	REGION B1.14.1 Transfer Unit
	    //// Transfer B1.14.1
	    #"B1.14.1"(TransferID := _."B1.14.1",
	               TransferSensor:=_."ASiGW-MCC001-bw143-C2: Input"."LoadPresence -B1.14.1",
	               Fault := DB_UDI.ProductionLine.Fault.Stop.Conveyor[_."B1.14.1"],
	               Upstream := DB_UDI.ProductionLine.Upstream.Conveyor[_."B1.14.1"],
	               FrontSensor:=_."ASiGW-MCC001-bw143-C2: Input"."FrontSensor -B1.14.1",
	               EndSensor:=_."ASiGW-MCC001-bw143-C2: Input"."EndSensor -B1.14.1",
	               "Left/RightSensor":=_."ASiGW-MCC001-bw143-C2: Input"."LeftSensor -B1.14.1",
	               Downstream := DB_UDI.ProductionLine.DownstreamAccu.Stop.Conveyor[_."B1.14.1"],
	               TransferDirection := DB_ToteTracking.Conveyor[_."B1.14.1"].ToteDir,
	               StartSignal => _."ASiGW-MCC001-bw143-C2: Output"."StartSignal -B1.14.1",
	               Cmd1 => _."ASiGW-MCC001-bw143-C2: Output"."Command1 -B1.14.1",
	               Cmd2 => _."ASiGW-MCC001-bw143-C2: Output"."Command2 -B1.14.1",
	               ErrorReset => _."ASiGW-MCC001-bw143-C2: Output"."ErrorReset -B1.14.1");

	END_REGION

	REGION B1.15.1
	    //// B1.15.1 (Go straight TR_B1.17.1)
	    #"B1.15.1"(ConveyorID := _."B1.15.1",
	               ConveyorSensor:=_."ASiGW-MCC001-bw143-C2: Input"."Sensor B1.15.1",
	               Fault := DB_UDI.ProductionLine.Fault.Stop.Conveyor[_."B1.15.1"],
	               Upstream := DB_UDI.ProductionLine.Upstream.Conveyor[_."B1.15.1"],
	               Downstream := DB_UDI.ProductionLine.DownstreamAccu.Stop.Conveyor[_."B1.15.1"],
	               Interlock := DB_UDI.ProductionLine.Interlock.Stop.Conveyor[_."B1.15.1"],
	               RunForward=>_."ASiGW-MCC001-bw143-C2: Output"."Motor B1.15.1",
	               WriteAsiDir=>_."ASiGW-MCC001-bw143-C2: Output"."Dir B1.15.1");

	END_REGION

	REGION B1.15.2
	    //B1.15.2
	    #"B1.15.2"(ConveyorID := _."B1.15.2",
	               ConveyorSensor:=_."ASiGW-MCC001-bw143-C2: Input"."Sensor B1.15.2",
	               Fault := DB_UDI.ProductionLine.Fault.Stop.Conveyor[_."B1.15.2"],
	               Upstream := DB_UDI.ProductionLine.Upstream.Conveyor[_."B1.15.2"],
	               Downstream := DB_UDI.ProductionLine.DownstreamAccu.Stop.Conveyor[_."B1.15.2"],
	               Interlock := DB_UDI.ProductionLine.Interlock.Stop.Conveyor[_."B1.15.2"],
	               RunForward=>_."ASiGW-MCC001-bw143-C2: Output"."Motor B1.15.2",
	               WriteAsiDir=>_."ASiGW-MCC001-bw143-C2: Output"."Dir B1.15.2");

	END_REGION

	REGION B1.16.1
	    //B1.16.1
	    #"B1.16.1"(ConveyorID := _."B1.16.1",
	               ConveyorSensor:=_."ASiGW-MCC001-bw143-C2: Input"."Sensor B1.16.8",
	               Fault := DB_UDI.ProductionLine.Fault.Stop.Conveyor[_."B1.16.1"],
	               Upstream := DB_UDI.ProductionLine.Upstream.Conveyor[_."B1.16.1"],
	               Downstream := DB_UDI.ProductionLine.DownstreamAccu.Stop.Conveyor[_."B1.16.1"],
	               Interlock := DB_UDI.ProductionLine.Interlock.Stop.Conveyor[_."B1.16.1"],
	               RunForward => _."ASiGW-MCC001-bw143-C2: Output"."Motor B1.16.1",
	               WriteAsiDir => _."ASiGW-MCC001-bw143-C2: Output"."Dir B1.16.1");

	END_REGION

	REGION B1.16.2
	    //B1.16.2
	    #"B1.16.2"(ConveyorID := _."B1.16.2",
	               ConveyorSensor:=_."ASiGW-MCC001-bw143-C2: Input"."Sensor B1.16.8",
	               Fault := DB_UDI.ProductionLine.Fault.Stop.Conveyor[_."B1.16.2"],
	               Upstream := DB_UDI.ProductionLine.Upstream.Conveyor[_."B1.16.2"],
	               Downstream := DB_UDI.ProductionLine.DownstreamAccu.Stop.Conveyor[_."B1.16.2"],
	               Interlock := DB_UDI.ProductionLine.Interlock.Stop.Conveyor[_."B1.16.2"],
	               RunForward=>_."ASiGW-MCC001-bw143-C2: Output"."Motor B1.16.2",
	               WriteAsiDir=>_."ASiGW-MCC001-bw143-C2: Output"."Dir B1.16.2");

	END_REGION

	REGION B1.16.3
	    //B1.16.3
	    #"B1.16.3"(ConveyorID := _."B1.16.3",
	               ConveyorSensor:=_."ASiGW-MCC001-bw143-C2: Input"."Sensor B1.16.8",
	               Fault := DB_UDI.ProductionLine.Fault.Stop.Conveyor[_."B1.16.3"],
	               Upstream := DB_UDI.ProductionLine.Upstream.Conveyor[_."B1.16.3"],
	               Downstream := DB_UDI.ProductionLine.DownstreamAccu.Stop.Conveyor[_."B1.16.3"],
	               Interlock := DB_UDI.ProductionLine.Interlock.Stop.Conveyor[_."B1.16.3"],
	               RunForward=>_."ASiGW-MCC001-bw143-C2: Output"."Motor B1.16.3",
	               WriteAsiDir=>_."ASiGW-MCC001-bw143-C2: Output"."Dir B1.16.3");

	END_REGION

	REGION B1.16.4
	    //B1.16.4
	    #"B1.16.4"(ConveyorID := _."B1.16.4",
	               ConveyorSensor:=_."ASiGW-MCC001-bw143-C2: Input"."Sensor B1.16.8",
	               Fault := DB_UDI.ProductionLine.Fault.Stop.Conveyor[_."B1.16.4"],
	               Upstream := DB_UDI.ProductionLine.Upstream.Conveyor[_."B1.16.4"],
	               Downstream := DB_UDI.ProductionLine.DownstreamAccu.Stop.Conveyor[_."B1.16.4"],
	               Interlock := DB_UDI.ProductionLine.Interlock.Stop.Conveyor[_."B1.16.4"],
	               RunForward=>_."ASiGW-MCC001-bw143-C2: Output"."Motor B1.16.4",
	               WriteAsiDir=>_."ASiGW-MCC001-bw143-C2: Output"."Dir B1.16.4");

	END_REGION

	REGION B1.16.5
	    //B1.16.5
	    #"B1.16.5"(ConveyorID := _."B1.16.5",
	               ConveyorSensor:=_."ASiGW-MCC001-bw143-C2: Input"."Sensor B1.16.8",
	               Fault := DB_UDI.ProductionLine.Fault.Stop.Conveyor[_."B1.16.5"],
	               Upstream := DB_UDI.ProductionLine.Upstream.Conveyor[_."B1.16.5"],
	               Downstream := DB_UDI.ProductionLine.DownstreamAccu.Stop.Conveyor[_."B1.16.5"],
	               Interlock := DB_UDI.ProductionLine.Interlock.Stop.Conveyor[_."B1.16.5"],
	               RunForward=>_."ASiGW-MCC001-bw143-C2: Output"."Motor B1.16.5",
	               WriteAsiDir=>_."ASiGW-MCC001-bw143-C2: Output"."Dir B1.16.5");

	END_REGION

	REGION B1.16.6
	    //B1.16.6
	    #"B1.16.6"(ConveyorID := _."B1.16.6",
	               ConveyorSensor:=_."ASiGW-MCC001-bw143-C2: Input"."Sensor B1.16.8",
	               Fault := DB_UDI.ProductionLine.Fault.Stop.Conveyor[_."B1.16.6"],
	               Upstream := DB_UDI.ProductionLine.Upstream.Conveyor[_."B1.16.6"],
	               Downstream := DB_UDI.ProductionLine.DownstreamAccu.Stop.Conveyor[_."B1.16.6"],
	               Interlock := DB_UDI.ProductionLine.Interlock.Stop.Conveyor[_."B1.16.6"],
	               RunForward=>_."ASiGW-MCC001-bw143-C2: Output"."Motor B1.16.6",
	               WriteAsiDir=>_."ASiGW-MCC001-bw143-C2: Output"."Dir B1.16.6");

	END_REGION

	REGION B1.16.7
	    //B1.16.7
	    #"B1.16.7"(ConveyorID := _."B1.16.7",
	               ConveyorSensor:=_."ASiGW-MCC001-bw143-C2: Input"."Sensor B1.16.8",
	               Fault := DB_UDI.ProductionLine.Fault.Stop.Conveyor[_."B1.16.7"],
	               Upstream := DB_UDI.ProductionLine.Upstream.Conveyor[_."B1.16.7"],
	               Downstream := DB_UDI.ProductionLine.DownstreamAccu.Stop.Conveyor[_."B1.16.7"],
	               Interlock := DB_UDI.ProductionLine.Interlock.Stop.Conveyor[_."B1.16.7"],
	               RunForward => _."ASiGW-MCC001-bw143-C2: Output"."Motor B1.16.7",
	               WriteAsiDir => _."ASiGW-MCC001-bw143-C2: Output"."Dir B1.16.7");

	END_REGION

	REGION B1.16.8
	    //B1.16.8
	    #"B1.16.8"(ConveyorID := _."B1.16.8",
	               ConveyorSensor:=_."ASiGW-MCC001-bw143-C2: Input"."Sensor B1.16.8",
	               Fault := DB_UDI.ProductionLine.Fault.Stop.Conveyor[_."B1.16.8"],
	               Upstream := DB_UDI.ProductionLine.Upstream.Conveyor[_."B1.16.8"],
	               Downstream := DB_UDI.ProductionLine.DownstreamAccu.Stop.Conveyor[_."B1.16.8"],
	               Interlock := DB_UDI.ProductionLine.Interlock.Stop.Conveyor[_."B1.16.8"],
	               RunForward=>_."ASiGW-MCC001-bw143-C2: Output"."Motor B1.16.8",
	               WriteAsiDir=>_."ASiGW-MCC001-bw143-C2: Output"."Dir B1.16.8");

	END_REGION

	REGION B1.17.1
	    //// B1.17.1 (DP3)
	    #"B1.17.1"(ConveyorID := _."B1.17.1",
	               ConveyorSensor:=_."ASiGW-MCC001-bw143-C2: Input"."Sensor B1.17.1",
	               Fault := DB_UDI.ProductionLine.Fault.Stop.Conveyor[_."B1.17.1"],
	               Upstream := DB_UDI.ProductionLine.Upstream.Conveyor[_."B1.17.1"],
	               Downstream := DB_UDI.ProductionLine.DownstreamAccu.Stop.Conveyor[_."B1.17.1"],
	               Interlock := DB_UDI.ProductionLine.Interlock.Stop.Conveyor[_."B1.17.1"],
	               RunForward => _."ASiGW-MCC001-bw143-C2: Output"."Motor B1.17.1",
	               WriteAsiDir => _."ASiGW-MCC001-bw143-C2: Output"."Dir B1.17.1");

	END_REGION

	REGION B1.17.2
	    //B1.17.2
	    #"B1.17.2"(ConveyorID := _."B1.17.2",
	               ConveyorSensor:=_."ASiGW-MCC001-bw143-C2: Input"."Sensor B1.17.2",
	               Fault := DB_UDI.ProductionLine.Fault.Stop.Conveyor[_."B1.17.2"],
	               Upstream := DB_UDI.ProductionLine.Upstream.Conveyor[_."B1.17.2"],
	               Downstream := DB_UDI.ProductionLine.DownstreamAccu.Stop.Conveyor[_."B1.17.2"],
	               Interlock := DB_UDI.ProductionLine.Interlock.Stop.Conveyor[_."B1.17.2"],
	               RunForward => _."ASiGW-MCC001-bw143-C2: Output"."Motor B1.17.2",
	               WriteAsiDir => _."ASiGW-MCC001-bw143-C2: Output"."Dir B1.17.2");

	END_REGION

	REGION B1.17.3
	    //B1.17.3
	    #"B1.17.3"(ConveyorID := _."B1.17.3",
	               ConveyorSensor:=_."ASiGW-MCC001-bw143-C2: Input"."Sensor B1.17.3",
	               Fault := DB_UDI.ProductionLine.Fault.Stop.Conveyor[_."B1.17.3"],
	               Upstream := DB_UDI.ProductionLine.Upstream.Conveyor[_."B1.17.3"],
	               Downstream := DB_UDI.ProductionLine.DownstreamAccu.Stop.Conveyor[_."B1.17.3"],
	               Interlock := DB_UDI.ProductionLine.Interlock.Stop.Conveyor[_."B1.17.3"],
	               RunForward => _."ASiGW-MCC001-bw143-C2: Output"."Motor B1.17.3",
	               WriteAsiDir => _."ASiGW-MCC001-bw143-C2: Output"."Dir B1.17.3");

	END_REGION

	REGION B1.17.4
	    //B1.17.4
	    #"B1.17.4"(ConveyorID := _."B1.17.4",
	               ConveyorSensor:=_."ASiGW-MCC001-bw143-C2: Input"."Sensor B1.17.4",
	               Fault := DB_UDI.ProductionLine.Fault.Stop.Conveyor[_."B1.17.4"],
	               Upstream := DB_UDI.ProductionLine.Upstream.Conveyor[_."B1.17.4"],
	               Downstream := DB_UDI.ProductionLine.DownstreamAccu.Stop.Conveyor[_."B1.17.4"],
	               Interlock := DB_UDI.ProductionLine.Interlock.Stop.Conveyor[_."B1.17.4"],
	               RunForward => _."ASiGW-MCC001-bw143-C2: Output"."Motor B1.17.4",
	               WriteAsiDir => _."ASiGW-MCC001-bw143-C2: Output"."Dir B1.17.4");

	END_REGION

	REGION B1.18.1 Transfer Unit
	    //// Transfer B1.18.1
	    #"B1.18.1"(TransferID := _."B1.18.1",
	               TransferSensor:=_."ASiGW-MCC001-bw143-C2: Input"."LoadPresence -B1.18.1",
	               Fault := DB_UDI.ProductionLine.Fault.Stop.Conveyor[_."B1.18.1"],
	               Upstream := DB_UDI.ProductionLine.Upstream.Conveyor[_."B1.18.1"],
	               FrontSensor:=_."ASiGW-MCC001-bw143-C2: Input"."FrontSensor -B1.18.1",
	               EndSensor:=_."ASiGW-MCC001-bw143-C2: Input"."EndSensor -B1.18.1",
	               "Left/RightSensor":=_."ASiGW-MCC001-bw143-C2: Input"."LeftSensor -B1.18.1",
	               Downstream := DB_UDI.ProductionLine.DownstreamAccu.Stop.Conveyor[_."B1.18.1"],
	               TransferDirection := DB_ToteTracking.Conveyor[_."B1.18.1"].ToteDir,
	               StartSignal => _."ASiGW-MCC001-bw143-C2: Output"."StartSignal -B1.18.1",
	               Cmd1 => _."ASiGW-MCC001-bw143-C2: Output"."Command1 -B1.18.1",
	               Cmd2 => _."ASiGW-MCC001-bw143-C2: Output"."Command2 -B1.18.1",
	               ErrorReset => _."ASiGW-MCC001-bw143-C2: Output"."ErrorReset -B1.18.1");

	END_REGION

	REGION B1.19.1
	    //B1.19.1
	    #"B1.19.1"(ConveyorID := _."B1.19.1",
	               ConveyorSensor:=_."ASiGW-MCC001-bw143-C2: Input"."Sensor B1.19.1",
	               Fault := DB_UDI.ProductionLine.Fault.Stop.Conveyor[_."B1.19.1"],
	               Upstream := DB_UDI.ProductionLine.Upstream.Conveyor[_."B1.19.1"],
	               Downstream := DB_UDI.ProductionLine.DownstreamAccu.Stop.Conveyor[_."B1.19.1"],
	               Interlock := DB_UDI.ProductionLine.Interlock.Stop.Conveyor[_."B1.19.1"],
	               RunForward => _."ASiGW-MCC001-bw143-C2: Output"."Motor B1.19.1",
	               WriteAsiDir => _."ASiGW-MCC001-bw143-C2: Output"."Dir B1.19.1");

	END_REGION

	REGION B1.20.1
	    //B1.20.1
	    #"B1.20.1"(ConveyorID := _."B1.20.1",
	               ConveyorSensor:=_."ASiGW-MCC001-bw143-C2: Input"."Sensor B1.20.1",
	               Fault := DB_UDI.ProductionLine.Fault.Stop.Conveyor[_."B1.20.1"],
	               Upstream := DB_UDI.ProductionLine.Upstream.Conveyor[_."B1.20.1"],
	               Downstream := DB_UDI.ProductionLine.DownstreamAccu.Stop.Conveyor[_."B1.20.1"],
	               Interlock := DB_UDI.ProductionLine.Interlock.Stop.Conveyor[_."B1.20.1"],
	               RunForward => _."ASiGW-MCC001-bw143-C2: Output"."Motor B1.20.1",
	               WriteAsiDir => _."ASiGW-MCC001-bw143-C2: Output"."Dir B1.20.1");

	END_REGION

	REGION B1.20.2
	    //B1.20.2
	    #"B1.20.2"(ConveyorID := _."B1.20.2",
	               ConveyorSensor:=_."ASiGW-MCC001-bw143-C2: Input"."Sensor B1.20.2",
	               Fault := DB_UDI.ProductionLine.Fault.Stop.Conveyor[_."B1.20.2"],
	               Upstream := DB_UDI.ProductionLine.Upstream.Conveyor[_."B1.20.2"],
	               Downstream := DB_UDI.ProductionLine.DownstreamAccu.Stop.Conveyor[_."B1.20.2"],
	               Interlock := DB_UDI.ProductionLine.Interlock.Stop.Conveyor[_."B1.20.2"],
	               RunForward => _."ASiGW-MCC001-bw143-C2: Output"."Motor B1.20.2",
	               WriteAsiDir => _."ASiGW-MCC001-bw143-C2: Output"."Dir B1.20.2");

	END_REGION

	REGION B1.21.1
	    //B1.21.1
	    #"B1.21.1"(ConveyorID := _."B1.21.1",
	               ConveyorSensor:=_."ASiGW-MCC001-bw143-C2: Input"."Sensor B1.21.1",
	               Fault := DB_UDI.ProductionLine.Fault.Stop.Conveyor[_."B1.21.1"],
	               Upstream := DB_UDI.ProductionLine.Upstream.Conveyor[_."B1.21.1"],
	               Downstream := DB_UDI.ProductionLine.DownstreamAccu.Stop.Conveyor[_."B1.21.1"],
	               Interlock := DB_UDI.ProductionLine.Interlock.Stop.Conveyor[_."B1.21.1"],
	               RunForward => _."ASiGW-MCC001-bw143-C2: Output"."Motor B1.21.1",
	               WriteAsiDir => _."ASiGW-MCC001-bw143-C2: Output"."Dir B1.21.1");

	END_REGION

	REGION B1.21.2
	    //B1.21.2
	    #"B1.21.2"(ConveyorID := _."B1.21.2",
	               ConveyorSensor:=_."ASiGW-MCC001-bw143-C2: Input"."Sensor B1.21.2",
	               Fault := DB_UDI.ProductionLine.Fault.Stop.Conveyor[_."B1.21.2"],
	               Upstream := DB_UDI.ProductionLine.Upstream.Conveyor[_."B1.21.2"],
	               Downstream := DB_UDI.ProductionLine.DownstreamAccu.Stop.Conveyor[_."B1.21.2"],
	               Interlock := DB_UDI.ProductionLine.Interlock.Stop.Conveyor[_."B1.21.2"],
	               RunForward => _."ASiGW-MCC001-bw143-C2: Output"."Motor B1.21.2",
	               WriteAsiDir => _."ASiGW-MCC001-bw143-C2: Output"."Dir B1.21.2");

	END_REGION

	REGION B1.21.3
	    //B1.21.3
	    #"B1.21.3"(ConveyorID := _."B1.21.3",
	               ConveyorSensor:=_."ASiGW-MCC001-bw143-C2: Input"."Sensor B1.23.1",
	               Fault := DB_UDI.ProductionLine.Fault.Stop.Conveyor[_."B1.21.3"],
	               Upstream := DB_UDI.ProductionLine.Upstream.Conveyor[_."B1.21.3"],
	               Downstream := DB_UDI.ProductionLine.DownstreamAccu.Stop.Conveyor[_."B1.21.3"],
	               Interlock := DB_UDI.ProductionLine.Interlock.Stop.Conveyor[_."B1.21.3"],
	               RunForward => _."ASiGW-MCC001-bw143-C2: Output"."Motor B1.21.3",
	               WriteAsiDir => _."ASiGW-MCC001-bw143-C2: Output"."Dir B1.21.3");

	END_REGION

	REGION B1.22.1
	    //B1.22.1
	    #"B1.22.1"(ConveyorID := _."B1.22.1",
	               ConveyorSensor:=_."ASiGW-MCC001-bw143-C2: Input"."Sensor B1.23.1",
	               Fault := DB_UDI.ProductionLine.Fault.Stop.Conveyor[_."B1.22.1"],
	               Upstream := DB_UDI.ProductionLine.Upstream.Conveyor[_."B1.22.1"],
	               Downstream := DB_UDI.ProductionLine.DownstreamAccu.Stop.Conveyor[_."B1.22.1"],
	               Interlock := DB_UDI.ProductionLine.Interlock.Stop.Conveyor[_."B1.22.1"],
	               RunForward => _."ASiGW-MCC001-bw143-C2: Output"."Motor - B1.22.1",
	               WriteAsiDir => _."ASiGW-MCC001-bw143-C2: Output"."2-30A Dir",
	               WriteAsiSpeed => _."ASiGW-MCC001-bw143-C2: Output"."2-30A Speed");

	END_REGION

	REGION B1.23.1
	    ////B1.23.1 Arm for Merger1
	    #"B1.23.1"(ConveyorID := _."B1.23.1",
	               ConveyorSensor:=_."ASiGW-MCC001-bw143-C2: Input"."Sensor B1.23.1",
	               Fault := DB_UDI.ProductionLine.Fault.Stop.Conveyor[_."B1.23.1"],
	               Upstream := DB_UDI.ProductionLine.Upstream.Conveyor[_."B1.23.1"],
	               Downstream := DB_UDI.ProductionLine.DownstreamAccu.Stop.Conveyor[_."B1.23.1"],
	               Interlock := DB_UDI.ProductionLine.Interlock.Stop.Conveyor[_."B1.23.1"],
	               RunForward => _."ASiGW-MCC001-bw143-C2: Output"."Motor B1.23.1",
	               WriteAsiDir => _."ASiGW-MCC001-bw143-C2: Output"."Dir B1.23.1");

	END_REGION

	REGION C1.3.1 Transfer Unit
	    ////Transfer C1.3.1
	    #"C1.3.1"(TransferID := _."C1.3.1",
	              TransferSensor:=_."ASiGW-MCC001-bw143-C2: Input"."LoadPresence -C1.3.1",
	              Fault := DB_UDI.ProductionLine.Fault.Stop.Conveyor[_."C1.3.1"],
	              Upstream := DB_UDI.ProductionLine.Upstream.Conveyor[_."C1.3.1"],
	              FrontSensor:=_."ASiGW-MCC001-bw143-C2: Input"."FrontSensor -C1.3.1",
	              EndSensor:=_."ASiGW-MCC001-bw143-C2: Input"."EndSensor -C1.3.1",
	              "Left/RightSensor":=_."ASiGW-MCC001-bw143-C2: Input"."LeftSensor -C1.3.1",
	              Downstream := DB_UDI.ProductionLine.DownstreamAccu.Stop.Conveyor[_."C1.3.1"],
	              TransferDirection := DB_ToteTracking.Conveyor[_."C1.3.1"].ToteDir,
	              StartSignal => _."ASiGW-MCC001-bw143-C2: Output"."StartSignal -C1.3.1",
	              Cmd1 => _."ASiGW-MCC001-bw143-C2: Output"."Command1 -C1.3.1",
	              Cmd2 => _."ASiGW-MCC001-bw143-C2: Output"."Command2 -C1.3.1",
	              ErrorReset => _."ASiGW-MCC001-bw143-C2: Output"."ErrorReset -C1.3.1");

	END_REGION

	REGION C1.2.2
	    //// C1.2.2  (Go Right TR_C1.1.3)
	    #"C1.2.2"(ConveyorID := _."C1.2.2",
	              ConveyorSensor:=_."ASiGW-MCC001-bw143-C2: Input"."Sensor C1.2.2",
	              Fault := DB_UDI.ProductionLine.Fault.Stop.Conveyor[_."C1.2.2"],
	              Upstream := DB_UDI.ProductionLine.Upstream.Conveyor[_."C1.2.2"],
	              Downstream := DB_UDI.ProductionLine.DownstreamAccu.Stop.Conveyor[_."C1.2.2"],
	              Interlock := DB_UDI.ProductionLine.Interlock.Stop.Conveyor[_."C1.2.2"],
	              RunForward=>_."ASiGW-MCC001-bw143-C2: Output"."Motor C1.2.2",
	              WriteAsiDir=>_."ASiGW-MCC001-bw143-C2: Output"."Dir C1.2.2");

	END_REGION

	REGION C1.2.1
	    //C1.2.1
	    #"C1.2.1"(ConveyorID := _."C1.2.1",
	              ConveyorSensor:=_."ASiGW-MCC001-bw143-C2: Input"."Sensor C1.2.1",
	              Fault := DB_UDI.ProductionLine.Fault.Stop.Conveyor[_."C1.2.1"],
	              Upstream := DB_UDI.ProductionLine.Upstream.Conveyor[_."C1.2.1"],
	              Downstream := DB_UDI.ProductionLine.DownstreamAccu.Stop.Conveyor[_."C1.2.1"],
	              Interlock := DB_UDI.ProductionLine.Interlock.Stop.Conveyor[_."C1.2.1"],
	              RunForward=>_."ASiGW-MCC001-bw143-C2: Output"."Motor C1.2.1",
	              WriteAsiDir=>_."ASiGW-MCC001-bw143-C2: Output"."Dir C1.2.1");

	END_REGION

	REGION C1.4.1
	    //// C1.4.1  (Go Left TR_C1.1.3)
	    #"C1.4.1"(ConveyorID := _."C1.4.1",
	              ConveyorSensor:=_."ASiGW-MCC001-bw143-C2: Input"."Sensor C1.4.1",
	              Fault := DB_UDI.ProductionLine.Fault.Stop.Conveyor[_."C1.4.1"],
	              Upstream := DB_UDI.ProductionLine.Upstream.Conveyor[_."C1.4.1"],
	              Downstream := DB_UDI.ProductionLine.DownstreamAccu.Stop.Conveyor[_."C1.4.1"],
	              Interlock := DB_UDI.ProductionLine.Interlock.Stop.Conveyor[_."C1.4.1"],
	              RunForward=>_."ASiGW-MCC001-bw143-C2: Output"."Motor C1.4.1",
	              WriteAsiDir=>_."ASiGW-MCC001-bw143-C2: Output"."Dir C1.4.1");

	END_REGION

	REGION C1.4.2
	    //C1.4.2
	    #"C1.4.2"(ConveyorID := _."C1.4.2",
	              ConveyorSensor:=_."ASiGW-MCC001-bw143-C2: Input"."Sensor C1.4.2",
	              Fault := DB_UDI.ProductionLine.Fault.Stop.Conveyor[_."C1.4.2"],
	              Upstream := DB_UDI.ProductionLine.Upstream.Conveyor[_."C1.4.2"],
	              Downstream := DB_UDI.ProductionLine.DownstreamAccu.Stop.Conveyor[_."C1.4.2"],
	              Interlock := DB_UDI.ProductionLine.Interlock.Stop.Conveyor[_."C1.4.2"],
	              RunForward=>_."ASiGW-MCC001-bw143-C2: Output"."Motor C1.4.2",
	              WriteAsiDir=>_."ASiGW-MCC001-bw143-C2: Output"."Dir C1.4.2");

	END_REGION

	REGION D1.1.1
	    ////  D1.1.1 (Go Right DP4)
	    #"D1.1.1"(ConveyorID := _."D1.1.1",
	              ConveyorSensor:=_."ASiGW-MCC001-bw200-C1: Input"."Sensor D1.2.1",
	              Fault := DB_UDI.ProductionLine.Fault.Stop.Conveyor[_."D1.1.1"],
	              Upstream := DB_UDI.ProductionLine.Upstream.Conveyor[_."D1.1.1"],
	              Downstream := DB_UDI.ProductionLine.DownstreamAccu.Stop.Conveyor[_."D1.1.1"],
	              Interlock := DB_UDI.ProductionLine.Interlock.Stop.Conveyor[_."D1.1.1"],
	              RunForward=>_."ASiGW-MCC001-bw200-C1: Output"."Motor D1.1.1",
	              WriteAsiDir=>_."ASiGW-MCC001-bw200-C1: Output"."Dir D1.1.1");

	END_REGION

	REGION D1.2.1
	    //D1.2.1
	    #"D1.2.1"(ConveyorID := _."D1.2.1",
	              ConveyorSensor:=_."ASiGW-MCC001-bw200-C1: Input"."Sensor D1.2.1",
	              Fault := DB_UDI.ProductionLine.Fault.Stop.Conveyor[_."D1.2.1"],
	              Upstream := DB_UDI.ProductionLine.Upstream.Conveyor[_."D1.2.1"],
	              Downstream := DB_UDI.ProductionLine.DownstreamAccu.Stop.Conveyor[_."D1.2.1"],
	              Interlock := DB_UDI.ProductionLine.Interlock.Stop.Conveyor[_."D1.2.1"],
	              RunForward=>_."ASiGW-MCC001-bw200-C1: Output"."Motor - D1.2.1",
	              WriteAsiDir=>_."ASiGW-MCC001-bw200-C1: Output"."1-2A Dir",
	              WriteAsiSpeed=>_."ASiGW-MCC001-bw200-C1: Output"."1-2A Speed");

	END_REGION

	REGION D1.3.1
	    //D1.3.1
	    #"D1.3.1"(ConveyorID := _."D1.3.1",
	              ConveyorSensor:=_."ASiGW-MCC001-bw200-C1: Input"."Sensor D1.3.1",
	              Fault := DB_UDI.ProductionLine.Fault.Stop.Conveyor[_."D1.3.1"],
	              Upstream := DB_UDI.ProductionLine.Upstream.Conveyor[_."D1.3.1"],
	              Downstream := DB_UDI.ProductionLine.DownstreamAccu.Stop.Conveyor[_."D1.3.1"],
	              Interlock := DB_UDI.ProductionLine.Interlock.Stop.Conveyor[_."D1.3.1"],
	              RunForward=>_."ASiGW-MCC001-bw200-C1: Output"."Motor - D1.3.1",
	              WriteAsiDir=>_."ASiGW-MCC001-bw200-C1: Output"."1-2A Dir",
	              WriteAsiSpeed=>_."ASiGW-MCC001-bw200-C1: Output"."1-2A Speed");

	END_REGION

	REGION D1.4.1
	    //D1.4.1
	    #"D1.4.1"(ConveyorID := _."D1.4.1",
	              ConveyorSensor:=_."ASiGW-MCC001-bw200-C1: Input"."Sensor D1.4.1",
	              Fault := DB_UDI.ProductionLine.Fault.Stop.Conveyor[_."D1.4.1"],
	              Upstream := DB_UDI.ProductionLine.Upstream.Conveyor[_."D1.4.1"],
	              Downstream := DB_UDI.ProductionLine.DownstreamAccu.Stop.Conveyor[_."D1.4.1"],
	              Interlock := DB_UDI.ProductionLine.Interlock.Stop.Conveyor[_."D1.4.1"],
	              RunForward=>_."ASiGW-MCC001-bw200-C1: Output"."Motor D1.4.1",
	              WriteAsiDir=>_."ASiGW-MCC001-bw200-C1: Output"."Dir D1.4.1");

	END_REGION

	REGION D1.5.1
	    //D1.5.1
	    #"D1.5.1"(ConveyorID := _."D1.5.1",
	              ConveyorSensor:=_."ASiGW-MCC001-bw200-C1: Input"."Sensor D1.5.1",
	              Fault := DB_UDI.ProductionLine.Fault.Stop.Conveyor[_."D1.5.1"],
	              Upstream := DB_UDI.ProductionLine.Upstream.Conveyor[_."D1.5.1"],
	              Downstream := DB_UDI.ProductionLine.DownstreamAccu.Stop.Conveyor[_."D1.5.1"],
	              Interlock := DB_UDI.ProductionLine.Interlock.Stop.Conveyor[_."D1.5.1"],
	              RunForward=>_."ASiGW-MCC001-bw200-C1: Output"."Motor - D1.5.1",
	              WriteAsiDir=>_."ASiGW-MCC001-bw200-C1: Output"."1-4A Dir",
	              WriteAsiSpeed=>_."ASiGW-MCC001-bw200-C1: Output"."1-4A Speed");

	END_REGION

	REGION D1.6.1
	    //D1.6.1
	    #"D1.6.1"(ConveyorID := _."D1.6.1",
	              ConveyorSensor:=_."ASiGW-MCC001-bw200-C1: Input"."Sensor D1.6.1",
	              Fault := DB_UDI.ProductionLine.Fault.Stop.Conveyor[_."D1.6.1"],
	              Upstream := DB_UDI.ProductionLine.Upstream.Conveyor[_."D1.6.1"],
	              Downstream := DB_UDI.ProductionLine.DownstreamAccu.Stop.Conveyor[_."D1.6.1"],
	              Interlock := DB_UDI.ProductionLine.Interlock.Stop.Conveyor[_."D1.6.1"],
	              RunForward=>_."ASiGW-MCC001-bw200-C1: Output"."Motor D1.6.1",
	              WriteAsiDir=>_."ASiGW-MCC001-bw200-C1: Output"."Dir D1.6.1");

	END_REGION

	REGION D1.7.1
	    //D1.7.1
	    #"D1.7.1"(ConveyorID := _."D1.7.1",
	              ConveyorSensor:=_."ASiGW-MCC001-bw200-C1: Input"."Sensor D1.7.10",
	              Fault := DB_UDI.ProductionLine.Fault.Stop.Conveyor[_."D1.7.1"],
	              Upstream := DB_UDI.ProductionLine.Upstream.Conveyor[_."D1.7.1"],
	              Downstream := DB_UDI.ProductionLine.DownstreamAccu.Stop.Conveyor[_."D1.7.1"],
	              Interlock := DB_UDI.ProductionLine.Interlock.Stop.Conveyor[_."D1.7.1"],
	              RunForward=>_."ASiGW-MCC001-bw200-C1: Output"."Motor D1.7.1",
	              WriteAsiDir=>_."ASiGW-MCC001-bw200-C1: Output"."Dir D1.7.1");

	END_REGION

	REGION D1.7.2
	    //D1.7.2
	    #"D1.7.2"(ConveyorID := _."D1.7.2",
	              ConveyorSensor:=_."ASiGW-MCC001-bw200-C1: Input"."Sensor D1.7.10",
	              Fault := DB_UDI.ProductionLine.Fault.Stop.Conveyor[_."D1.7.2"],
	              Upstream := DB_UDI.ProductionLine.Upstream.Conveyor[_."D1.7.2"],
	              Downstream := DB_UDI.ProductionLine.DownstreamAccu.Stop.Conveyor[_."D1.7.2"],
	              Interlock := DB_UDI.ProductionLine.Interlock.Stop.Conveyor[_."D1.7.2"],
	              RunForward=>_."ASiGW-MCC001-bw200-C1: Output"."Motor D1.7.2",
	              WriteAsiDir=>_."ASiGW-MCC001-bw200-C1: Output"."Dir D1.7.2");

	END_REGION

	REGION D1.7.3
	    //D1.7.3
	    #"D1.7.3"(ConveyorID := _."D1.7.3",
	              ConveyorSensor:=_."ASiGW-MCC001-bw200-C1: Input"."Sensor D1.7.10",
	              Fault := DB_UDI.ProductionLine.Fault.Stop.Conveyor[_."D1.7.3"],
	              Upstream := DB_UDI.ProductionLine.Upstream.Conveyor[_."D1.7.3"],
	              Downstream := DB_UDI.ProductionLine.DownstreamAccu.Stop.Conveyor[_."D1.7.3"],
	              Interlock := DB_UDI.ProductionLine.Interlock.Stop.Conveyor[_."D1.7.3"],
	              RunForward=>_."ASiGW-MCC001-bw200-C1: Output"."Motor D1.7.3",
	              WriteAsiDir=>_."ASiGW-MCC001-bw200-C1: Output"."Dir D1.7.3");

	END_REGION

	REGION D1.7.4
	    //D1.7.4
	    #"D1.7.4"(ConveyorID := _."D1.7.4",
	              ConveyorSensor:=_."ASiGW-MCC001-bw200-C1: Input"."Sensor D1.7.10",
	              Fault := DB_UDI.ProductionLine.Fault.Stop.Conveyor[_."D1.7.4"],
	              Upstream := DB_UDI.ProductionLine.Upstream.Conveyor[_."D1.7.4"],
	              Downstream := DB_UDI.ProductionLine.DownstreamAccu.Stop.Conveyor[_."D1.7.4"],
	              Interlock := DB_UDI.ProductionLine.Interlock.Stop.Conveyor[_."D1.7.4"],
	              RunForward=>_."ASiGW-MCC001-bw200-C1: Output"."Motor D1.7.4",
	              WriteAsiDir=>_."ASiGW-MCC001-bw200-C1: Output"."Dir D1.7.4");

	END_REGION

	REGION D1.7.5
	    //D1.7.5
	    #"D1.7.5"(ConveyorID := _."D1.7.5",
	              ConveyorSensor:=_."ASiGW-MCC001-bw200-C1: Input"."Sensor D1.7.10",
	              Fault := DB_UDI.ProductionLine.Fault.Stop.Conveyor[_."D1.7.5"],
	              Upstream := DB_UDI.ProductionLine.Upstream.Conveyor[_."D1.7.5"],
	              Downstream := DB_UDI.ProductionLine.DownstreamAccu.Stop.Conveyor[_."D1.7.5"],
	              Interlock := DB_UDI.ProductionLine.Interlock.Stop.Conveyor[_."D1.7.5"],
	              RunForward=>_."ASiGW-MCC001-bw200-C1: Output"."Motor D1.7.5",
	              WriteAsiDir=>_."ASiGW-MCC001-bw200-C1: Output"."Dir D1.7.5");

	END_REGION

	REGION D1.7.6
	    //D1.7.6
	    #"D1.7.6"(ConveyorID := _."D1.7.6",
	              ConveyorSensor:=_."ASiGW-MCC001-bw200-C1: Input"."Sensor D1.7.10",
	              Fault := DB_UDI.ProductionLine.Fault.Stop.Conveyor[_."D1.7.6"],
	              Upstream := DB_UDI.ProductionLine.Upstream.Conveyor[_."D1.7.6"],
	              Downstream := DB_UDI.ProductionLine.DownstreamAccu.Stop.Conveyor[_."D1.7.6"],
	              Interlock := DB_UDI.ProductionLine.Interlock.Stop.Conveyor[_."D1.7.6"],
	              RunForward=>_."ASiGW-MCC001-bw200-C1: Output"."Motor D1.7.6",
	              WriteAsiDir=>_."ASiGW-MCC001-bw200-C1: Output"."Dir D1.7.6");

	END_REGION

	REGION D1.7.7
	    //D1.7.7
	    #"D1.7.7"(ConveyorID := _."D1.7.7",
	              ConveyorSensor:=_."ASiGW-MCC001-bw200-C1: Input"."Sensor D1.7.10",
	              Fault := DB_UDI.ProductionLine.Fault.Stop.Conveyor[_."D1.7.7"],
	              Upstream := DB_UDI.ProductionLine.Upstream.Conveyor[_."D1.7.7"],
	              Downstream := DB_UDI.ProductionLine.DownstreamAccu.Stop.Conveyor[_."D1.7.7"],
	              Interlock := DB_UDI.ProductionLine.Interlock.Stop.Conveyor[_."D1.7.7"],
	              RunForward => _."ASiGW-MCC001-bw200-C1: Output"."Motor D1.7.7",
	              WriteAsiDir => _."ASiGW-MCC001-bw200-C1: Output"."Dir D1.7.7");

	END_REGION

	REGION D1.7.8
	    //D1.7.8
	    #"D1.7.8"(ConveyorID := _."D1.7.8",
	              ConveyorSensor:=_."ASiGW-MCC001-bw200-C1: Input"."Sensor D1.7.10",
	              Fault := DB_UDI.ProductionLine.Fault.Stop.Conveyor[_."D1.7.8"],
	              Upstream := DB_UDI.ProductionLine.Upstream.Conveyor[_."D1.7.8"],
	              Downstream := DB_UDI.ProductionLine.DownstreamAccu.Stop.Conveyor[_."D1.7.8"],
	              Interlock := DB_UDI.ProductionLine.Interlock.Stop.Conveyor[_."D1.7.8"],
	              RunForward=>_."ASiGW-MCC001-bw200-C1: Output"."Motor D1.7.8",
	              WriteAsiDir=>_."ASiGW-MCC001-bw200-C1: Output"."Dir D1.7.8");

	END_REGION

	REGION D1.7.9
	    //D1.7.9
	    #"D1.7.9"(ConveyorID := _."D1.7.9",
	              ConveyorSensor:=_."ASiGW-MCC001-bw200-C1: Input"."Sensor D1.7.10",
	               Fault := DB_UDI.ProductionLine.Fault.Stop.Conveyor[_."D1.7.9"],
	               Upstream := DB_UDI.ProductionLine.Upstream.Conveyor[_."D1.7.9"],
	               Downstream := DB_UDI.ProductionLine.DownstreamAccu.Stop.Conveyor[_."D1.7.9"],
	               Interlock := DB_UDI.ProductionLine.Interlock.Stop.Conveyor[_."D1.7.9"],
	               RunForward=>_."ASiGW-MCC001-bw200-C1: Output"."Motor D1.7.9",
	               WriteAsiDir=>_."ASiGW-MCC001-bw200-C1: Output"."Dir D1.7.9");

	END_REGION

	REGION D1.7.10
	    //D1.7.10
	    #"D1.7.10"(ConveyorID := _."D1.7.10",
	               ConveyorSensor:=_."ASiGW-MCC001-bw200-C1: Input"."Sensor D1.7.10",
	               Fault := DB_UDI.ProductionLine.Fault.Stop.Conveyor[_."D1.7.10"],
	               Upstream := DB_UDI.ProductionLine.Upstream.Conveyor[_."D1.7.10"],
	               Downstream := DB_UDI.ProductionLine.DownstreamAccu.Stop.Conveyor[_."D1.7.10"],
	               Interlock := DB_UDI.ProductionLine.Interlock.Stop.Conveyor[_."D1.7.10"],
	               RunForward => _."ASiGW-MCC001-bw200-C1: Output"."Motor D1.7.10",
	               WriteAsiDir => _."ASiGW-MCC001-bw200-C1: Output"."Dir D1.7.10");

	END_REGION

	REGION D1.8.1
	    //D1.8.1
	    #"D1.8.1"(ConveyorID := _."D1.8.1",
	              ConveyorSensor:=_."ASiGW-MCC001-bw200-C1: Input"."Sensor D1.8.1",
	              Fault := DB_UDI.ProductionLine.Fault.Stop.Conveyor[_."D1.8.1"],
	              Upstream := DB_UDI.ProductionLine.Upstream.Conveyor[_."D1.8.1"],
	              Downstream := DB_UDI.ProductionLine.DownstreamAccu.Stop.Conveyor[_."D1.8.1"],
	              Interlock := DB_UDI.ProductionLine.Interlock.Stop.Conveyor[_."D1.8.1"],
	              RunForward => _."ASiGW-MCC001-bw200-C1: Output"."Motor D1.8.1",
	              WriteAsiDir => _."ASiGW-MCC001-bw200-C1: Output"."Dir D1.8.1");

	END_REGION

	REGION D1.8.2
	    //D1.8.2
	    #"D1.8.2"(ConveyorID := _."D1.8.2",
	              ConveyorSensor:=_."ASiGW-MCC001-bw200-C1: Input"."Sensor D1.8.2",
	              Fault := DB_UDI.ProductionLine.Fault.Stop.Conveyor[_."D1.8.2"],
	              Upstream := DB_UDI.ProductionLine.Upstream.Conveyor[_."D1.8.2"],
	              Downstream := DB_UDI.ProductionLine.DownstreamAccu.Stop.Conveyor[_."D1.8.2"],
	              Interlock := DB_UDI.ProductionLine.Interlock.Stop.Conveyor[_."D1.8.2"],
	              RunForward => _."ASiGW-MCC001-bw200-C1: Output"."Motor D1.8.2",
	              WriteAsiDir => _."ASiGW-MCC001-bw200-C1: Output"."Dir D1.8.2");

	END_REGION

	REGION D1.8.3
	    //D1.8.3
	    #"D1.8.3"(ConveyorID := _."D1.8.3",
	              ConveyorSensor:=_."ASiGW-MCC001-bw200-C1: Input"."Sensor D1.8.3",
	              Fault := DB_UDI.ProductionLine.Fault.Stop.Conveyor[_."D1.8.3"],
	              Upstream := DB_UDI.ProductionLine.Upstream.Conveyor[_."D1.8.3"],
	              Downstream := DB_UDI.ProductionLine.DownstreamAccu.Stop.Conveyor[_."D1.8.3"],
	              Interlock := DB_UDI.ProductionLine.Interlock.Stop.Conveyor[_."D1.8.3"],
	              RunForward => _."ASiGW-MCC001-bw200-C1: Output"."Motor D1.8.3",
	              WriteAsiDir => _."ASiGW-MCC001-bw200-C1: Output"."Dir D1.8.3");

	END_REGION

	REGION D1.9.1 Transfer Unit
	    ////Transfer D1.9.1
	    #"D1.9.2"(TransferID := _."D1.9.1",
	              TransferSensor:=_."ASiGW-MCC001-bw200-C1: Input"."LoadPresence -D1.9.1",
	              Fault := DB_UDI.ProductionLine.Fault.Stop.Conveyor[_."D1.9.1"],
	              Upstream := DB_UDI.ProductionLine.Upstream.Conveyor[_."D1.9.1"],
	              FrontSensor:=_."ASiGW-MCC001-bw200-C1: Input"."FrontSensor -D1.9.1",
	              EndSensor:=_."ASiGW-MCC001-bw200-C1: Input"."EndSensor -D1.9.1",
	              "Left/RightSensor":=_."ASiGW-MCC001-bw200-C1: Input"."LeftSensor -D1.9.1",
	              Downstream := DB_UDI.ProductionLine.DownstreamAccu.Stop.Conveyor[_."D1.9.1"],
	              TransferDirection := DB_ToteTracking.Conveyor[_."D1.9.1"].ToteDir,
	              StartSignal => _."ASiGW-MCC001-bw200-C1: Output"."StartSignal -D1.9.1",
	              Cmd1 =>  _."ASiGW-MCC001-bw200-C1: Output"."Command1 -D1.9.1",
	              Cmd2 => _."ASiGW-MCC001-bw200-C1: Output"."Command2 -D1.9.1",
	              ErrorReset =>  _."ASiGW-MCC001-bw200-C1: Output"."ErrorReset -D1.9.1");

	END_REGION

	REGION D1.10.1 Transfer Unit
	    ////Transfer D1.10.1
	    #"D1.10.1"(TransferID := _."D1.10.1",
	              Fault := DB_UDI.ProductionLine.Fault.Stop.Conveyor[_."D1.10.1"],
	              Upstream := DB_UDI.ProductionLine.Upstream.Conveyor[_."D1.10.1"],
	              Downstream := DB_UDI.ProductionLine.DownstreamAccu.Stop.Conveyor[_."D1.10.1"],
	              TransferDirection := DB_ToteTracking.Conveyor[_."D1.10.1"].ToteDir,
	              StartSignal =>  _."ASiGW-MCC001-bw200-C1: Output"."StartSignal -D1.10.1",
	              Cmd1 =>  _."ASiGW-MCC001-bw200-C1: Output"."Command1 -D1.10.1",
	              Cmd2 =>  _."ASiGW-MCC001-bw200-C1: Output"."Command2 -D1.10.1",
	              ErrorReset =>  _."ASiGW-MCC001-bw200-C1: Output"."ErrorReset -D1.10.1");

	END_REGION

	REGION D1.11.1
	    //D1.11.1
	    #"D1.11.1"(ConveyorID := _."D1.11.1",
	               ConveyorSensor:=_."ASiGW-MCC001-bw200-C1: Input"."Sensor D1.11.1",
	               Fault := DB_UDI.ProductionLine.Fault.Stop.Conveyor[_."D1.11.1"],
	               Upstream := DB_UDI.ProductionLine.Upstream.Conveyor[_."D1.11.1"],
	               Downstream := DB_UDI.ProductionLine.DownstreamAccu.Stop.Conveyor[_."D1.11.1"],
	               Interlock := DB_UDI.ProductionLine.Interlock.Stop.Conveyor[_."D1.11.1"],
	               RunForward => _."ASiGW-MCC001-bw200-C1: Output"."Motor D1.11.1",
	               WriteAsiDir => _."ASiGW-MCC001-bw200-C1: Output"."Dir D1.11.1");

	END_REGION

	REGION D1.11.2
	    //D1.11.2
	    #"D1.11.2"(ConveyorID := _."D1.11.2",
	               ConveyorSensor:=_."ASiGW-MCC001-bw200-C1: Input"."Sensor D1.11.2",
	               Fault := DB_UDI.ProductionLine.Fault.Stop.Conveyor[_."D1.11.2"],
	               Upstream := DB_UDI.ProductionLine.Upstream.Conveyor[_."D1.11.2"],
	               Downstream := DB_UDI.ProductionLine.DownstreamAccu.Stop.Conveyor[_."D1.11.2"],
	               Interlock := DB_UDI.ProductionLine.Interlock.Stop.Conveyor[_."D1.11.2"],
	               RunForward => _."ASiGW-MCC001-bw200-C1: Output"."Motor D1.11.2",
	               WriteAsiDir => _."ASiGW-MCC001-bw200-C1: Output"."Dir D1.11.2");

	END_REGION

	REGION D1.11.3
	    //D1.11.3
	    #"D1.11.3"(ConveyorID := _."D1.11.3",
	               ConveyorSensor:=_."ASiGW-MCC001-bw200-C1: Input"."Sensor D1.11.3",
	               Fault := DB_UDI.ProductionLine.Fault.Stop.Conveyor[_."D1.11.3"],
	               Upstream := DB_UDI.ProductionLine.Upstream.Conveyor[_."D1.11.3"],
	               Downstream := DB_UDI.ProductionLine.DownstreamAccu.Stop.Conveyor[_."D1.11.3"],
	               Interlock := DB_UDI.ProductionLine.Interlock.Stop.Conveyor[_."D1.11.3"],
	               RunForward => _."ASiGW-MCC001-bw200-C1: Output"."Motor D1.11.3",
	               WriteAsiDir => _."ASiGW-MCC001-bw200-C1: Output"."Dir D1.11.3");

	END_REGION

	REGION D1.12.1
	    //D1.12.1
	    #"D1.12.1"(ConveyorID := _."D1.12.1",
	               ConveyorSensor:=_."ASiGW-MCC001-bw200-C1: Input"."Sensor D1.12.3",
	               Fault := DB_UDI.ProductionLine.Fault.Stop.Conveyor[_."D1.12.1"],
	               Upstream := DB_UDI.ProductionLine.Upstream.Conveyor[_."D1.12.1"],
	               Downstream := DB_UDI.ProductionLine.DownstreamAccu.Stop.Conveyor[_."D1.12.1"],
	               Interlock := DB_UDI.ProductionLine.Interlock.Stop.Conveyor[_."D1.12.1"],
	               RunForward=>_."ASiGW-MCC001-bw200-C1: Output"."Motor D1.12.1",
	               WriteAsiDir=>_."ASiGW-MCC001-bw200-C1: Output"."Dir D1.12.1");

	END_REGION

	REGION D1.12.2
	    //D1.12.2
	    #"D1.12.2"(ConveyorID := _."D1.12.2",
	               ConveyorSensor:=_."ASiGW-MCC001-bw200-C1: Input"."Sensor D1.12.3",
	               Fault := DB_UDI.ProductionLine.Fault.Stop.Conveyor[_."D1.12.2"],
	               Upstream := DB_UDI.ProductionLine.Upstream.Conveyor[_."D1.12.2"],
	               Downstream := DB_UDI.ProductionLine.DownstreamAccu.Stop.Conveyor[_."D1.12.2"],
	               Interlock := DB_UDI.ProductionLine.Interlock.Stop.Conveyor[_."D1.12.2"],
	               RunForward => _."ASiGW-MCC001-bw200-C1: Output"."Motor D1.12.2",
	               WriteAsiDir => _."ASiGW-MCC001-bw200-C1: Output"."Dir D1.12.2");

	END_REGION

	REGION D1.12.3
	    ////End
	    #"D1.12.3"(ConveyorID := _."D1.12.3",
	               ConveyorSensor:=_."ASiGW-MCC001-bw200-C1: Input"."Sensor D1.12.3",
	               Fault := DB_UDI.ProductionLine.Fault.Stop.Conveyor[_."D1.12.3"],
	               Upstream := DB_UDI.ProductionLine.Upstream.Conveyor[_."D1.12.3"],
	               Downstream := DB_UDI.ProductionLine.DownstreamAccu.Stop.Conveyor[_."D1.12.3"],
	               Interlock := DB_UDI.ProductionLine.Interlock.Stop.Conveyor[_."D1.12.3"],
	               RunForward => _."ASiGW-MCC001-bw200-C1: Output"."Motor D1.12.3",
	               WriteAsiDir => _."ASiGW-MCC001-bw200-C1: Output"."Dir D1.12.3");

	END_REGION

	REGION E1.1.1
	    //E1.1.1
	    #"E1.1.1"(ConveyorID := _."E1.1.1",
	              ConveyorSensor:=_."ASiGW-MCC001-bw200-C1: Input"."Sensor E1.1.1",
	              Fault := DB_UDI.ProductionLine.Fault.Stop.Conveyor[_."E1.1.1"],
	              Upstream := DB_UDI.ProductionLine.Upstream.Conveyor[_."E1.1.1"],
	              Downstream := DB_UDI.ProductionLine.DownstreamAccu.Stop.Conveyor[_."E1.1.1"],
	              Interlock := DB_UDI.ProductionLine.Interlock.Stop.Conveyor[_."E1.1.1"],
	              RunForward=>_."ASiGW-MCC001-bw200-C1: Output"."Motor E1.1.1",
	              WriteAsiDir=>_."ASiGW-MCC001-bw200-C1: Output"."Dir E1.1.1");

	END_REGION

	REGION E1.1.2
	    //E1.1.2
	    #"E1.1.2"(ConveyorID := _."E1.1.2",
	              ConveyorSensor:=_."ASiGW-MCC001-bw200-C1: Input"."Sensor E1.1.4",
	              Fault := DB_UDI.ProductionLine.Fault.Stop.Conveyor[_."E1.1.2"],
	              Upstream := DB_UDI.ProductionLine.Upstream.Conveyor[_."E1.1.2"],
	              Downstream := DB_UDI.ProductionLine.DownstreamAccu.Stop.Conveyor[_."E1.1.2"],
	              Interlock := DB_UDI.ProductionLine.Interlock.Stop.Conveyor[_."E1.1.2"],
	              RunForward=>_."ASiGW-MCC001-bw200-C1: Output"."Motor E1.1.2",
	              WriteAsiDir=>_."ASiGW-MCC001-bw200-C1: Output"."Dir E1.1.2");

	END_REGION

	REGION E1.1.3
	    //E1.1.3
	    #"E1.1.3"(ConveyorID := _."E1.1.3",
	              ConveyorSensor:=_."ASiGW-MCC001-bw200-C1: Input"."Sensor E1.1.4",
	              Fault := DB_UDI.ProductionLine.Fault.Stop.Conveyor[_."E1.1.3"],
	              Upstream := DB_UDI.ProductionLine.Upstream.Conveyor[_."E1.1.3"],
	              Downstream := DB_UDI.ProductionLine.DownstreamAccu.Stop.Conveyor[_."E1.1.3"],
	              Interlock := DB_UDI.ProductionLine.Interlock.Stop.Conveyor[_."E1.1.3"],
	              RunForward=>_."ASiGW-MCC001-bw200-C1: Output"."Motor E1.1.3",
	              WriteAsiDir=>_."ASiGW-MCC001-bw200-C1: Output"."Dir E1.1.3");

	END_REGION

	REGION E1.1.4
	    //E1.1.4
	    #"E1.1.4"(ConveyorID := _."E1.1.4",
	              ConveyorSensor:=_."ASiGW-MCC001-bw200-C1: Input"."Sensor E1.1.4",
	              Fault := DB_UDI.ProductionLine.Fault.Stop.Conveyor[_."E1.1.4"],
	              Upstream := DB_UDI.ProductionLine.Upstream.Conveyor[_."E1.1.4"],
	              Downstream := DB_UDI.ProductionLine.DownstreamAccu.Stop.Conveyor[_."E1.1.4"],
	              Interlock := DB_UDI.ProductionLine.Interlock.Stop.Conveyor[_."E1.1.4"],
	              RunForward=>_."ASiGW-MCC001-bw200-C1: Output"."Motor E1.1.4",
	              WriteAsiDir=>_."ASiGW-MCC001-bw200-C1: Output"."Dir E1.1.4");

	END_REGION

	REGION E1.2.1
	    //E1.2.1
	    #"E1.2.1"(ConveyorID := _."E1.2.1",
	              ConveyorSensor:=_."ASiGW-MCC001-bw200-C1: Input"."Sensor E1.2.1",
	              Fault := DB_UDI.ProductionLine.Fault.Stop.Conveyor[_."E1.2.1"],
	              Upstream := DB_UDI.ProductionLine.Upstream.Conveyor[_."E1.2.1"],
	              Downstream := DB_UDI.ProductionLine.DownstreamAccu.Stop.Conveyor[_."E1.2.1"],
	              Interlock := DB_UDI.ProductionLine.Interlock.Stop.Conveyor[_."E1.2.1"],
	              RunForward=>_."ASiGW-MCC001-bw200-C1: Output"."Motor - E1.2.1",
	              WriteAsiDir=>_."ASiGW-MCC001-bw200-C1: Output"."1-21A Dir",
	              WriteAsiSpeed=>_."ASiGW-MCC001-bw200-C1: Output"."1-21A Speed");

	END_REGION

	REGION E1.3.1
	    //E1.3.1
	    #"E1.3.1"(ConveyorID := _."E1.3.1",
	              ConveyorSensor:=_."ASiGW-MCC001-bw200-C1: Input"."Sensor E1.3.1",
	              Fault := DB_UDI.ProductionLine.Fault.Stop.Conveyor[_."E1.3.1"],
	              Upstream := DB_UDI.ProductionLine.Upstream.Conveyor[_."E1.3.1"],
	              Downstream := DB_UDI.ProductionLine.DownstreamAccu.Stop.Conveyor[_."E1.3.1"],
	              Interlock := DB_UDI.ProductionLine.Interlock.Stop.Conveyor[_."E1.3.1"],
	              RunForward=>_."ASiGW-MCC001-bw200-C1: Output"."Motor - E1.3.1",
	              WriteAsiDir=>_."ASiGW-MCC001-bw200-C1: Output"."1-21A Dir",
	              WriteAsiSpeed=>_."ASiGW-MCC001-bw200-C1: Output"."1-21A Speed");

	END_REGION

	REGION E1.4.1
	    //E1.4.1
	    #"E1.4.1"(ConveyorID := _."E1.4.1",
	              ConveyorSensor:=_."ASiGW-MCC001-bw200-C1: Input"."Sensor E1.4.1",
	              Fault := DB_UDI.ProductionLine.Fault.Stop.Conveyor[_."E1.4.1"],
	              Upstream := DB_UDI.ProductionLine.Upstream.Conveyor[_."E1.4.1"],
	              Downstream := DB_UDI.ProductionLine.DownstreamAccu.Stop.Conveyor[_."E1.4.1"],
	              Interlock := DB_UDI.ProductionLine.Interlock.Stop.Conveyor[_."E1.4.1"],
	              RunForward=>_."ASiGW-MCC001-bw200-C1: Output"."Motor E1.4.1",
	              WriteAsiDir=>_."ASiGW-MCC001-bw200-C1: Output"."Dir E1.4.1");

	END_REGION

	REGION E1.5.1
	    //E1.5.1
	    #"E1.5.1"(ConveyorID := _."E1.5.1",
	              ConveyorSensor := _."ASiGW-MCC001-bw200-C1: Input"."Sensor E1.5.1",
	              Fault := DB_UDI.ProductionLine.Fault.Stop.Conveyor[_."E1.5.1"],
	              Upstream := DB_UDI.ProductionLine.Upstream.Conveyor[_."E1.5.1"],
	              Downstream := DB_UDI.ProductionLine.DownstreamAccu.Stop.Conveyor[_."E1.5.1"],
	              Interlock := DB_UDI.ProductionLine.Interlock.Stop.Conveyor[_."E1.5.1"],
	              RunForward => _."ASiGW-MCC001-bw200-C1: Output"."Motor - E1.5.1",
	              WriteAsiDir => _."ASiGW-MCC001-bw200-C1: Output"."1-23A Dir",
	              WriteAsiSpeed => _."ASiGW-MCC001-bw200-C1: Output"."1-23A Speed");


	END_REGION

	REGION E1.6.1
	    ////E1.6.1 Arm for Merger2
	    #"E1.6.1"(ConveyorID := _."E1.6.1",
	              ConveyorSensor:=_."ASiGW-MCC001-bw200-C1: Input"."Sensor E1.5.1",
	              Fault := DB_UDI.ProductionLine.Fault.Stop.Conveyor[_."E1.6.1"],
	              Upstream := DB_UDI.ProductionLine.Upstream.Conveyor[_."E1.6.1"],
	              Downstream := DB_UDI.ProductionLine.DownstreamAccu.Stop.Conveyor[_."E1.6.1"],
	              Interlock := DB_UDI.ProductionLine.Interlock.Stop.Conveyor[_."E1.6.1"],
	              RunForward=>_."ASiGW-MCC001-bw200-C1: Output"."Motor E1.6.1",
	              WriteAsiDir=>_."ASiGW-MCC001-bw200-C1: Output"."Dir E1.6.1");

	END_REGION


END_FUNCTION_BLOCK
END_NAMESPACE

